SUBAPPLICATION A2X_TO_QXA2 (* Ein gebuendeltes unidirektionales A2X (UP/DOWN) auf 2 physische logiBUS-Digitalausgaenge entbuendelt: A2X_2X_TO_2AX spaltet das Paar unmittelbar vor den beiden logiBUS_QXA-Ausgaengen auf 2 einzelne AX-Signale auf - 'SUB style': das Entbuendeln steckt im Composite, nicht in der Resource des Geraets. *)
  (* Standard: 61499-2; Description: Copyright (c) 2026 HR Agrartechnik GmbH This program and the accompanying materials are made available under the terms of the Eclipse Public License 2.0 which is available at https://www.eclipse.org/legal/epl-2.0/ SPDX-License-Identifier: EPL-2.0 *)
  (* Version 1.0, 2026-09-05, Franz Höpfinger, HR Agrartechnik GmbH, initial API and implementation and/or initial documentation *)
  PACKAGE MyLib::sys;
  IMPORT logiBUS::io::DQ::logiBUS_DO::Invalid;
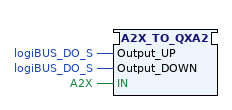
  VAR_INPUT
    Output_UP : logiBUS::io::DQ::logiBUS_DO_S := Invalid; (* Physischer Ausgang fuer forward/up *)
    Output_DOWN : logiBUS::io::DQ::logiBUS_DO_S := Invalid; (* Physischer Ausgang fuer backward/down *)
  END_VAR
  SOCKETS
    IN : adapter::types::unidirectional::A2X; (* Gebuendeltes UP/DOWN Eingangssignal *)
  END_SOCKETS
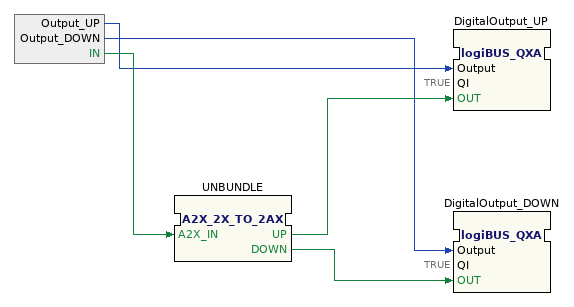
  FBS
    UNBUNDLE : adapter::conversion::unidirectional::A2X_2X_TO_2AX;
    DigitalOutput_UP : logiBUS::io::DQ::logiBUS_QXA(QI := TRUE);
    DigitalOutput_DOWN : logiBUS::io::DQ::logiBUS_QXA(QI := TRUE);
  END_FBS
  DATA_CONNECTIONS
    Output_UP TO DigitalOutput_UP.Output;
    Output_DOWN TO DigitalOutput_DOWN.Output;
  END_CONNECTIONS
  ADAPTER_CONNECTIONS
    IN TO UNBUNDLE.A2X_IN;
    UNBUNDLE.UP TO DigitalOutput_UP.OUT;
    UNBUNDLE.DOWN TO DigitalOutput_DOWN.OUT;
  END_CONNECTIONS
END_SUBAPPLICATION
